{attribute 'qualified_only'}
{attribute 'strict'}
TYPE eBetriebszustand :
(
	off, //nicht Betriebsbereit 
	error, //Fehlerbehafteter Stop(Sicherheitssteuerung)
	setup, //Wartung 
	warning, // Nicht fehlerbehafteter geplanter Stop 
	init, //Herstellung Betriebsbereitschaft 
	ready, //betriebsbereit 
	production, //Im Betrieb
	done, //Betrieb abgschlossen
	stop //geplanter Stillstand 
);
END_TYPE

(* stored: Version 1.1.0.1, ProductVersion 3.1.4024.15
   DUT eBetriebszustand: Id {aea1b32f-fa93-4aff-a081-8549f6ca8dfa} *)
